// TIA Portal project "babu_WaterFountainHMI" (V15)

(* hardware
DEVICE "S7-1200 station_1"  S7-1200 Station
   slot 0: "Rack_0"  S7-1200 Rack  Rack  V1.0
   slot 1: "PLC_1"  CPU 1214C DC/DC/DC  6ES7 214-1AG40-0XB0  V4.2
DEVICE "HMI_1"  KTP400 Basic PN
   slot 0: "HMI_1"  KTP400 Basic PN  6AV2 123-2DB03-0AX0  15.0.0.0
   slot 1: "HMI_RT_1"  KTP400 Basic PN  6AV2 123-2DB03-0AX0  15.0.0.0
   slot 5: "HMI_1.IE_CP_1"  PROFINET Interface  15.0.0.0
      slot 1: "PROFINET Interface_1"  PROFINET Interface
         slot 1: "Port_1"  Port
*)

// ===== PLC "PLC_1"  CPU 1214C DC/DC/DC =====

VAR_GLOBAL   // PLC tag table "Default tag table"
   "START PUSH BUTTON" AT %M0.0 : Bool;
   "Fountain Pump" AT %Q0.0 : Bool;
   "Fountain Pump Mem" AT %M0.1 : Bool;
   "STOP PUSH BUTTON" AT %M0.2 : Bool;
   "WATER SENSOR" AT %M0.3 : Bool;
   "TEMP" AT %M0.4 : Bool;
   "WATER SENSOR MEM" AT %M0.5 : Bool;
   "WATER SENSOR MEM OUT" AT %M0.6 : Bool;
END_VAR

// folder: System blocks/Program resources

DATA_BLOCK "IEC_Timer_0_DB"   // DB1
{ S7_Optimized_Access := 'TRUE' }
AUTHOR : Simatic
FAMILY : IEC
NAME : IEC_TMR
VERSION : 1.0
// stored: InstanceOfName IEC_TIMER
"IEC_TIMER"
BEGIN
END_DATA_BLOCK

// folder: (top level)

ORGANIZATION_BLOCK "Main"   // OB1, LAD, ProgramCycle
TITLE = "Main Program Sweep (Cycle)"
{ S7_Optimized_Access := 'TRUE' }
VERSION : 0.1
   VAR_INPUT
      Initial_Call : Bool;   // Initial call of this OB
      Remanence : Bool;   // =True, if remanent data are available
   END_VAR
   VAR_TEMP   // added for the SCL form of the ladder/FBD networks
      _w1 : Bool;
   END_VAR
BEGIN

REGION Network 1
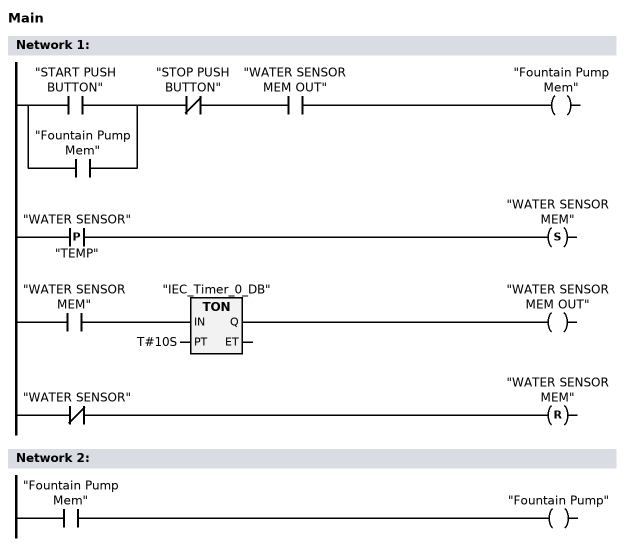
   "Fountain Pump Mem" := ("START PUSH BUTTON" OR "Fountain Pump Mem") AND NOT "STOP PUSH BUTTON" AND "WATER SENSOR MEM OUT";
   #_w1 := "WATER SENSOR" AND NOT "TEMP";   // rising edge of "WATER SENSOR"
   "TEMP" := "WATER SENSOR";
   IF #_w1 THEN "WATER SENSOR MEM" := TRUE; END_IF;
   "IEC_Timer_0_DB".TON(IN := "WATER SENSOR MEM", PT := T#10S);
   "WATER SENSOR MEM OUT" := "IEC_Timer_0_DB".Q;
   IF NOT "WATER SENSOR" THEN "WATER SENSOR MEM" := FALSE; END_IF;
END_REGION

REGION Network 2
   RUNG wire#powerrail
      Contact( "Fountain Pump Mem" )
      Coil( "Fountain Pump" )
   END_RUNG
   // the same network as SCL:
   "Fountain Pump" := "Fountain Pump Mem";
END_REGION
END_ORGANIZATION_BLOCK

(* ===== HMI "HMI_RT_1" =====
connection "HMI_Connection_1": ETHERNET, SMART_S7_1200_OMS

HMI tags "Default tag table"
   "START PUSH BUTTON" : Bool = PLC "START PUSH BUTTON" AT %M0.0, 1 s
   "STOP PUSH BUTTON" : Bool = PLC "STOP PUSH BUTTON" AT %M0.2, 1 s
   "Fountain Pump" : Bool = PLC "Fountain Pump" AT %Q0.0, 1 s

screen "Root screen" 480x272, template "Template_1"
   Switch "Pushbutton_Round_R" at 18,70 size 50x50; CaptionText 'Switch'; TextOff '0'; TextOn '1'; PictureOff "Pushbutton_Round_R_Off_256c"; PictureOn "Pushbutton_Round_R_On_256c"
      ProcessValue <- "STOP PUSH BUTTON"
   Switch "Pushbutton_Round_G" at 18,9 size 50x50; CaptionText 'Switch'; TextOff '0'; TextOn '1'; PictureOff "Pushbutton_Round_G_Off_256c"; PictureOn "Pushbutton_Round_G_On_256c"
      ProcessValue <- "START PUSH BUTTON"
   Circle "Circle_1" at 380,30 size 48x48
      Appearance <- "Fountain Pump"
   TextField "Text field_1" at 353,9 size 92x17; Text 'Water Fountain'
*)